{attribute 'qualified_only'}
{attribute 'strict'}
{attribute 'to_string'}
TYPE E_GearCommand : (
		Idle := 0,
		Enable,
		Disable,
		GearInStationary,
		GearInVelocity,
		GearInPosition
	);
END_TYPE

(* stored: Version 1.1.0.1
   DUT E_GearCommand: Id {fee1741e-425e-4ae1-b586-6be04bf3b35e} *)
